FUNCTION_BLOCK EL2034
VAR
	{attribute addProperty Name "WcState"}
	_wcState : WcStateInputToggle;
	{attribute addProperty Name "Info data"}
	_infoData : InfoDataBase;
	_io : EL2034_Data;
END_VAR

PROPERTY IO : REFERENCE TO EL2034_Data
GET
IO REF= _io;
END_GET
END_PROPERTY

PROPERTY WcState : REFERENCE TO WcStateInputToggle
GET
WcState REF= _wcState;
END_GET
END_PROPERTY

END_FUNCTION_BLOCK

(* stored: Version 1.1.0.1, ProductVersion 3.1.4024.9
   POU EL2034: Id {ccdf7fb1-6280-0a59-08e8-0c889268391b}, SpecialFunc None
   Property IO: Id {041fb26d-4b6b-07c3-2e1f-6449b0cec665}
   Get Get: Id {11a21d2f-d60c-0cd1-2b62-8248e27d7e15}
   Property WcState: Id {f3c4aa76-06bb-0166-01b5-baa9938a40db}
   Get Get: Id {096e9518-0804-03a7-23b3-42ac9e0b9390} *)
